# EPICS substitutions: IOCs/MS_DAQ/iocBoot/iocMS_TwoThetaStep/MS_TwoThetaStep.substitutions
file "$(TOP)/db/MS.db"
{
pattern
{P, R, BeamEnergy, Current, ShutterOne, ShutterTwo, StopperStatus, ExposureTime, Images, ImageName, ImagePath, isAcquiring, Acquiring, DS, DSUser, SEDTop, PilatusServerUser, PilatusServer, DataPath, TestDataPath, DetDataPath,}
{MS:, twoTheta:, SR-DI:getBeamEnergy, SRC01-DI-DCCT1:getDcctCurrent, I09FE-VA-PSH:getStatus, I09OH-VA-PSH:getStatus, I09FE-PSS-PHST:getStatus, I09-ES-CAM1:setExpTime, I09-ES-CAM1:setNImages, I09-ES-CAM1:setImageName, I09-ES-CAM1:setImgPath, I09-ES-CAM1:isAcquring, I09-ES-CAM1:acquire, 10.1.14.100, dcasu, /PETRA/SED, det, 10.3.3.8, /home/control/MS-XPD-ScanTool/DATA, MS/testDevData, /home/det/images,}
}

file "$(TOP)/db/MS_TwoThetaStep.db"
{
pattern
{P,   R,         twoTheta,                       twoThetaSpeed,						  Spinner,                        SampleContainer,}
{MS:, twoTheta:, I09R2-MO-MC3:ES-DIFF-STP-ROTX2, I09R2-MO-MC3:ES-DIFF-STP-ROTX2.VELO, I09R2-MO-MC1:ES-DIFF-STP-ROTX3, I09R2-MO-MC1:ES-DIFF-STP-ROTX1,}
}
